FUNCTION_BLOCK PUBLIC Converters_TestSuit EXTENDS TcUnit.FB_TestSuite
VAR
END_VAR

CheckSource_To_DestinationWithBool();

// todo, all other tests

METHOD PUBLIC CheckSource_To_DestinationWithBool
VAR
	in : BOOL := TRUE;
	_BOOL : BOOL;
	_BYTE : BYTE;
	_DATE : DATE;
	_DINT : DINT;
	_DT : DT;
	_DWORD : DWORD;
	_INT : INT;
	_LINT : LINT;
	_LREAL : LREAL;
	_LWORD : LWORD;
	_REAL : REAL;
	_SINT : SINT;
	_STRING : STRING;
	_TIME : TIME;
	_TOD : TOD;
	_UDINT : UDINT;
	_UINT : UINT;
	_ULINT : ULINT;
	_USINT : USINT;
	_WORD : WORD;
END_VAR
TEST('CheckSource_To_DestinationWithBool');

// @TEST-FIXTURE

// @TEST-RUN
Convert_Source_TO_Destination(in,_BOOL);
Convert_Source_TO_Destination(in,_BYTE);

// @TEST-ASSSERT
AssertTrue(
	Condition := (_BOOL = in),
	Message := 'BOOL incorrectly converted'
);

AssertTrue(
	Condition := (_BYTE = BOOL_TO_BYTE(in)),
	Message := 'BYTE incorrectly converted'
);

TEST_FINISHED();
END_METHOD

END_FUNCTION_BLOCK

(* stored: Version 1.1.0.1, ProductVersion 3.1.4024.12
   POU Converters_TestSuit: Id {4d30f73e-9617-42a5-9076-ace59b4cbdde}, SpecialFunc None
   Method CheckSource_To_DestinationWithBool: Id {d19bf4d4-3869-07ac-0ec8-00d77588470a} *)
